TYPE ST_Bridge_TSCS_INPUTS :
// 	Inputs from bridge terminal (bridge with TSCS PLC)
STRUCT
	TSCS_Byte : ARRAY [0..4] OF BYTE;		// Boolean words from TSCS PLC (5x 8 Booleans)
	
	TDU_TestSignal_RB : UDINT;				// Diagnostic signal readback TDU->TSCS->TDU
END_STRUCT
END_TYPE

(* stored: Version 1.1.0.1, ProductVersion 3.1.4024.6
   DUT ST_Bridge_TSCS_INPUTS: Id {7d2aed18-8bf0-4a0d-adc6-fa69b66256b7} *)
